PROGRAM UR3_Robot
VAR
	iniciar_secuencia_1 : BOOL;

	pos_separator_ok : BOOL;
	vi_get_img : BOOL ;
	estado_cabezal :INT;
	cabezal :BOOL;
	vi_img_ok : BOOL;
	i : BOOL;
	
	giro_cabezal :REAL;

	cx : REAL;
	cy : REAL;
	turn : REAL;
	cabezal_retirado :BOOL;
	regresar : BOOL;
	vi_image_proces: BOOL; 
	poner_cabeza : BOOL;
	
	vi_img_cabezal_dere_ok : BOOL;
	vi_img_cabezal_dere_proc_ok : BOOL;
	vi_get_img_cabezal_dere : BOOL;


END_VAR

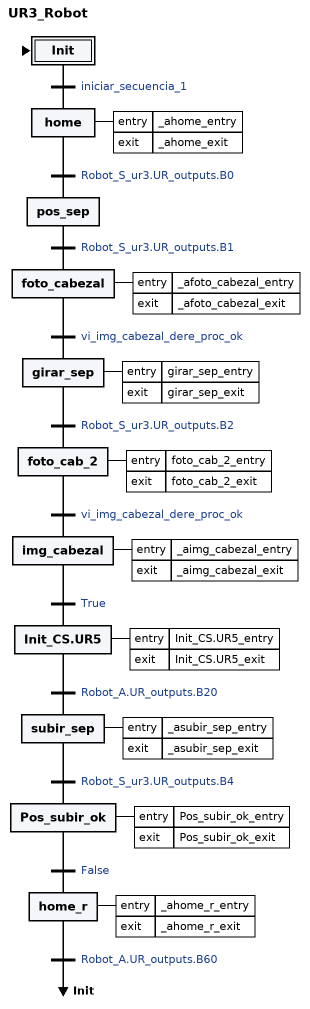
INITIAL_STEP Init:
END_STEP
TRANSITION FROM Init TO home
    := iniciar_secuencia_1;
END_TRANSITION
STEP home:
    _ahome_entry(P1);  // entry action
    _ahome_exit(P0);  // exit action
END_STEP
TRANSITION FROM home TO pos_sep
    := Robot_S_ur3.UR_outputs.B0;
END_TRANSITION
STEP pos_sep:
END_STEP
TRANSITION FROM pos_sep TO foto_cabezal
    := Robot_S_ur3.UR_outputs.B1;
END_TRANSITION
STEP foto_cabezal:
    _afoto_cabezal_entry(P1);  // entry action
    _afoto_cabezal_exit(P0);  // exit action
END_STEP
TRANSITION FROM foto_cabezal TO girar_sep
    := vi_img_cabezal_dere_proc_ok;
END_TRANSITION
STEP girar_sep:
    girar_sep_entry(P1);  // entry action
    girar_sep_exit(P0);  // exit action
END_STEP
TRANSITION FROM girar_sep TO foto_cab_2
    := Robot_S_ur3.UR_outputs.B2;
END_TRANSITION
STEP foto_cab_2:
    foto_cab_2_entry(P1);  // entry action
    foto_cab_2_exit(P0);  // exit action
END_STEP
TRANSITION FROM foto_cab_2 TO img_cabezal
    := vi_img_cabezal_dere_proc_ok;
END_TRANSITION
STEP img_cabezal:
    _aimg_cabezal_entry(P1);  // entry action
    _aimg_cabezal_exit(P0);  // exit action
END_STEP
TRANSITION FROM img_cabezal TO Init_CS_UR5
    := True;
END_TRANSITION
STEP Init_CS_UR5:  // name as stored: Init_CS.UR5
    Init_CS.UR5_entry(P1);  // entry action
    Init_CS.UR5_exit(P0);  // exit action
END_STEP
TRANSITION FROM Init_CS_UR5 TO subir_sep
    := Robot_A.UR_outputs.B20;
END_TRANSITION
STEP subir_sep:
    _asubir_sep_entry(P1);  // entry action
    _asubir_sep_exit(P0);  // exit action
END_STEP
TRANSITION FROM subir_sep TO Pos_subir_ok
    := Robot_S_ur3.UR_outputs.B4;
END_TRANSITION
STEP Pos_subir_ok:
    Pos_subir_ok_entry(P1);  // entry action
    Pos_subir_ok_exit(P0);  // exit action
END_STEP
TRANSITION FROM Pos_subir_ok TO home_r
    := False;
END_TRANSITION
STEP home_r:
    _ahome_r_entry(P1);  // entry action
    _ahome_r_exit(P0);  // exit action
END_STEP
TRANSITION FROM home_r TO Init
    := Robot_A.UR_outputs.B60;
END_TRANSITION

ACTION _afoto_cabezal_entry:
vi_get_img_cabezal_dere := TRUE;
END_ACTION

ACTION _afoto_cabezal_exit:
vi_get_img_cabezal_dere := FALSE;
vi_img_cabezal_dere_proc_ok := FALSE;
data_to_robot.head_roll_left := turn;
END_ACTION

ACTION _ahome_entry:
Robot_S_ur3.UR_inputs.Bits.B0 := TRUE;
END_ACTION

ACTION _ahome_exit:
Robot_S_ur3.UR_inputs.Bits.B0 := False;
END_ACTION

ACTION _ahome_r_entry:
Robot_A.UR_inputs.Bits.B27 := TRUE;
regresar := False;
END_ACTION

ACTION _ahome_r_exit:
Robot_A.UR_inputs.Bits.B27 := False;
END_ACTION

ACTION _aimg_cabezal_entry:
pos_separator_ok := TRUE;
END_ACTION

ACTION _aimg_cabezal_exit:
pos_separator_ok := False;
END_ACTION

ACTION _asubir_sep_entry:
Robot_S_ur3.UR_inputs.Bits.B20 := TRUE;
END_ACTION

ACTION _asubir_sep_exit:
Robot_S_ur3.UR_inputs.Bits.B20 := FALSE;
END_ACTION

ACTION foto_cab_2_entry:
vi_get_img_cabezal_dere := TRUE;
END_ACTION

ACTION foto_cab_2_exit:
vi_get_img_cabezal_dere := FALSE;
vi_img_cabezal_dere_proc_ok := FALSE;
data_to_robot.head_roll_right := turn;
END_ACTION

ACTION girar_sep_entry:
Robot_S_ur3.UR_inputs.Bits.B0 := TRUE;
END_ACTION

ACTION girar_sep_exit:
Robot_S_ur3.UR_inputs.Bits.B0 := False;
END_ACTION

ACTION Init_UR5_entry:
RCts.RCts.UR5_robot.iniciar := True;
END_ACTION

ACTION Init_UR5_exit:
RCts.RCts.UR5_robot.iniciar := False;
END_ACTION

ACTION Pos_subir_ok_entry:
Robot_A.UR_inputs.Bits.B20 := TRUE;
END_ACTION

ACTION Pos_subir_ok_exit:
Robot_A.UR_inputs.Bits.B20 := False;
END_ACTION

END_PROGRAM

(* stored: Version 1.1.0.1, ProductVersion 3.1.4024.4
   POU UR3_Robot: Id {236ed89c-461a-4e2f-b21a-6543ee10a66c}, SpecialFunc None
   Action _afoto_cabezal_entry: Id {52f1c111-13ab-4549-8874-541c02f261dc}
   Action _afoto_cabezal_exit: Id {f37b2425-3923-4fdf-89ff-2f253b619ede}
   Action _ahome_entry: Id {71ce866c-fa91-4c36-a857-c17e1612e479}
   Action _ahome_exit: Id {4747ef67-74d2-486c-9203-4c28f94e5182}
   Action _ahome_r_entry: Id {5d59ec00-15a9-4251-87e9-db795aa72728}
   Action _ahome_r_exit: Id {70df0f93-16aa-447b-acff-d27f0ef73eae}
   Action _aimg_cabezal_entry: Id {3fe36791-3a39-4c57-b00a-0e720157059e}
   Action _aimg_cabezal_exit: Id {49914240-5f76-4790-81c9-38182204a047}
   Action _asubir_sep_entry: Id {835eb47f-8faf-41ce-8056-9d07ce7d7020}
   Action _asubir_sep_exit: Id {974f9616-705a-4b20-8dbb-738e80ec17f0}
   Action foto_cab_2_entry: Id {25015224-b57f-4421-bdab-87fac59770ae}
   Action foto_cab_2_exit: Id {d9901155-bf7b-4323-a34e-75ba417c4cbc}
   Action girar_sep_entry: Id {76c39167-d352-4e45-9816-aad54382be21}
   Action girar_sep_exit: Id {dc96bd1e-fa34-4679-9311-270a1aaa7e08}
   Action Init_UR5_entry: Id {1e8f29fe-fc49-4c67-9e0f-db1c1848fa7f}
   Action Init_UR5_exit: Id {544214e9-6f93-4ebd-8905-83c236daf4db}
   Action Pos_subir_ok_entry: Id {cd034212-a1b0-4d5f-b99d-ca0c1afbf9de}
   Action Pos_subir_ok_exit: Id {f71d015b-6f4b-4eb9-8bf9-44dee863e6b3} *)
